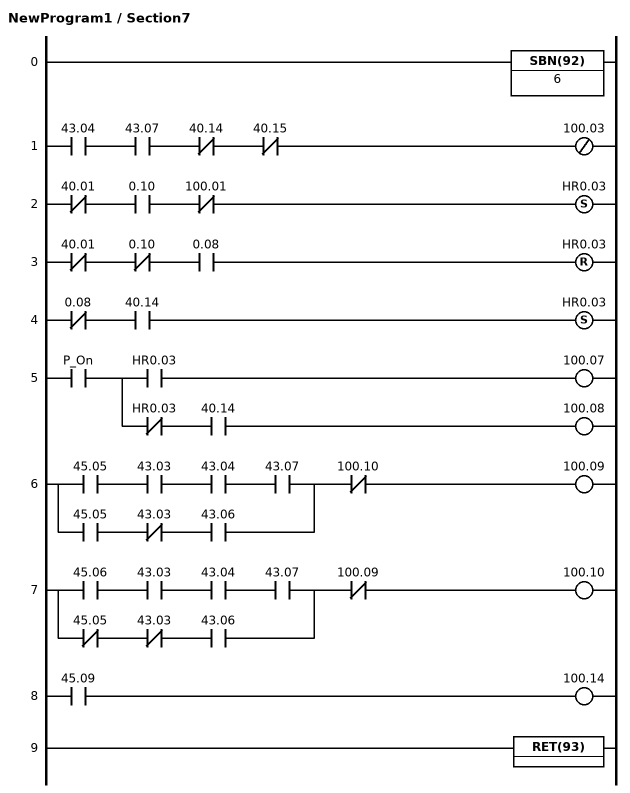
; [picture p24: NewProgram1 / Section7, rungs 0-9]
; rung 0
SBN(92) 6
; rung 1
LD 43.04
AND 43.07
ANDNOT 40.14
ANDNOT 40.15
OUTNOT 100.03
; rung 2
LDNOT 40.01
AND 0.10
ANDNOT 100.01
SET HR0.03
; rung 3
LDNOT 40.01
ANDNOT 0.10
AND 0.08
RSET HR0.03
; rung 4
LDNOT 0.08
AND 40.14
SET HR0.03
; rung 5
LD P_On
OUT TR0
AND HR0.03
OUT 100.07
LD TR0
ANDNOT HR0.03
AND 40.14
OUT 100.08
; rung 6
LD 45.05
AND 43.03
AND 43.04
AND 43.07
LD 45.05
ANDNOT 43.03
AND 43.06
ORLD
ANDNOT 100.10
OUT 100.09
; rung 7
LD 45.06
AND 43.03
AND 43.04
AND 43.07
LDNOT 45.05
ANDNOT 43.03
AND 43.06
ORLD
ANDNOT 100.09
OUT 100.10
; rung 8
LD 45.09
OUT 100.14
; rung 9
RET(93)

### Section Section8

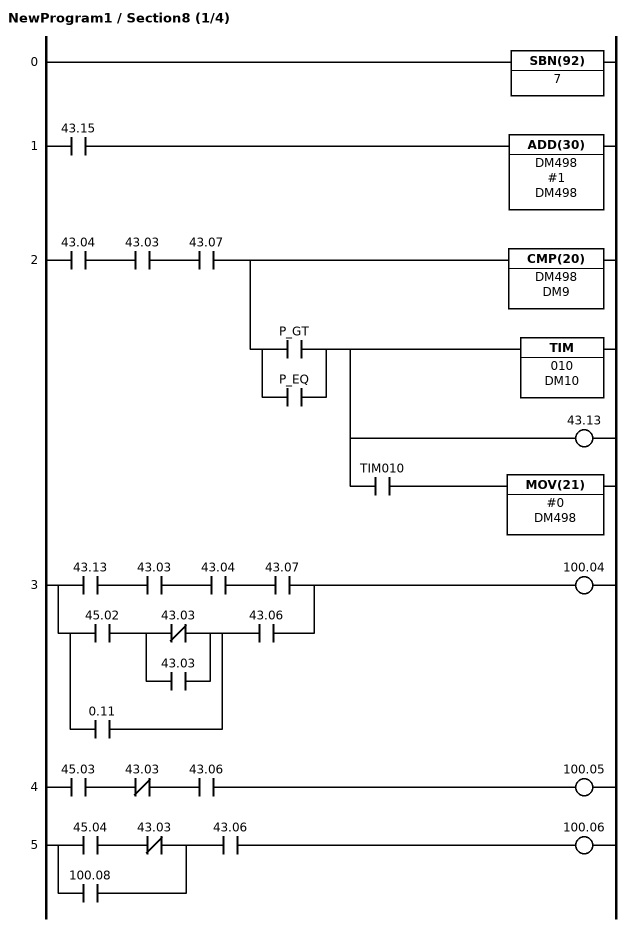
; rung 0
SBN(92) 7
; rung 1
LD 43.15
ADD(30) DM498 #1 DM498
; rung 2
LD 43.04
AND 43.03
AND 43.07
CMP(20) DM498 DM9
LD P_GT
OR P_EQ
ANDLD
TIM 010 DM10
OUT 43.13
AND TIM010
MOV(21) #0 DM498
; rung 3
LD 43.13
AND 43.03
AND 43.04
AND 43.07
LD 45.02
LDNOT 43.03
OR 43.03
ANDLD
OR 0.11
AND 43.06
ORLD
OUT 100.04
; rung 4
LD 45.03
ANDNOT 43.03
AND 43.06
OUT 100.05
; rung 5
LD 45.04
ANDNOT 43.03
OR 100.08
AND 43.06
OUT 100.06

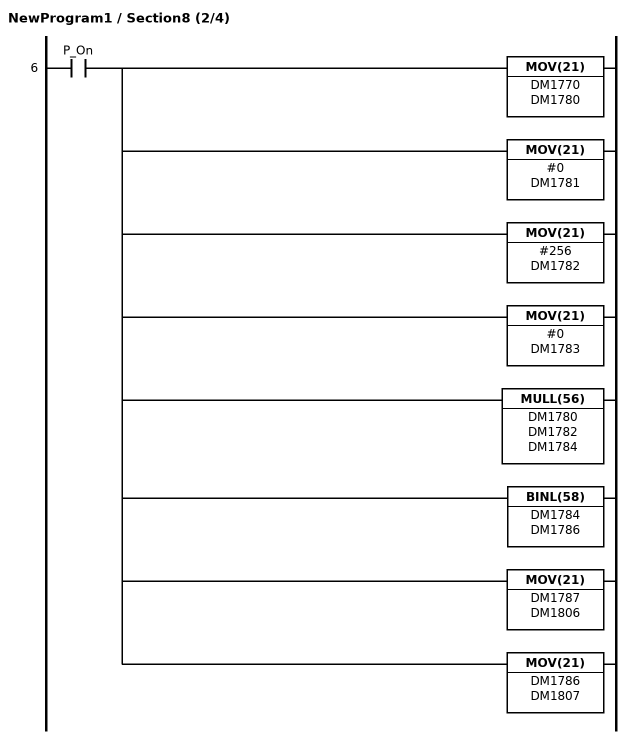
; rung 6
LD P_On
MOV(21) DM1770 DM1780
MOV(21) #0 DM1781
MOV(21) #256 DM1782
MOV(21) #0 DM1783
MULL(56) DM1780 DM1782 DM1784
BINL(58) DM1784 DM1786
MOV(21) DM1787 DM1806
MOV(21) DM1786 DM1807

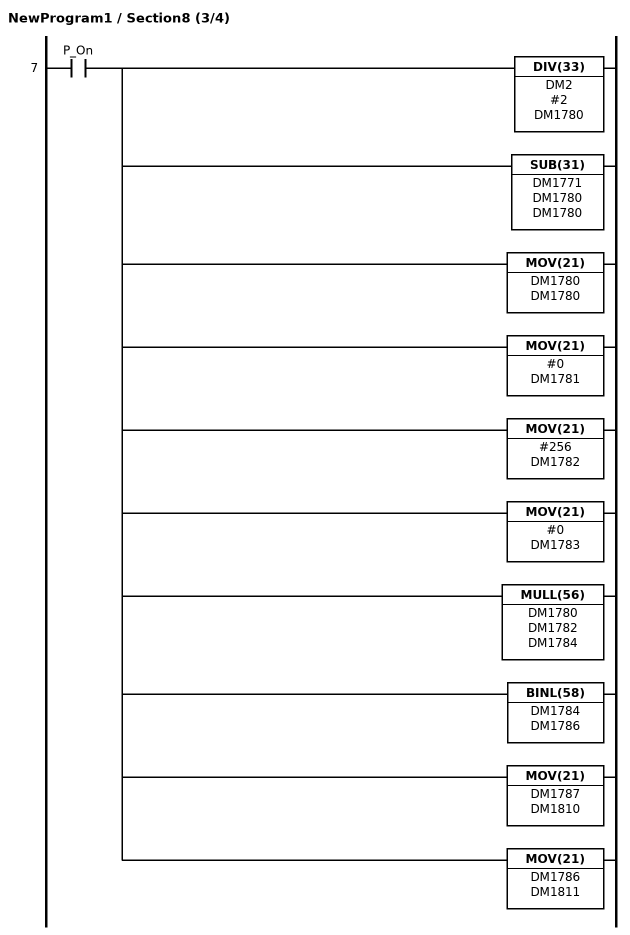
; rung 7
LD P_On
DIV(33) DM2 #2 DM1780
SUB(31) DM1771 DM1780 DM1780
MOV(21) DM1780 DM1780
MOV(21) #0 DM1781
MOV(21) #256 DM1782
MOV(21) #0 DM1783
MULL(56) DM1780 DM1782 DM1784
BINL(58) DM1784 DM1786
MOV(21) DM1787 DM1810
MOV(21) DM1786 DM1811

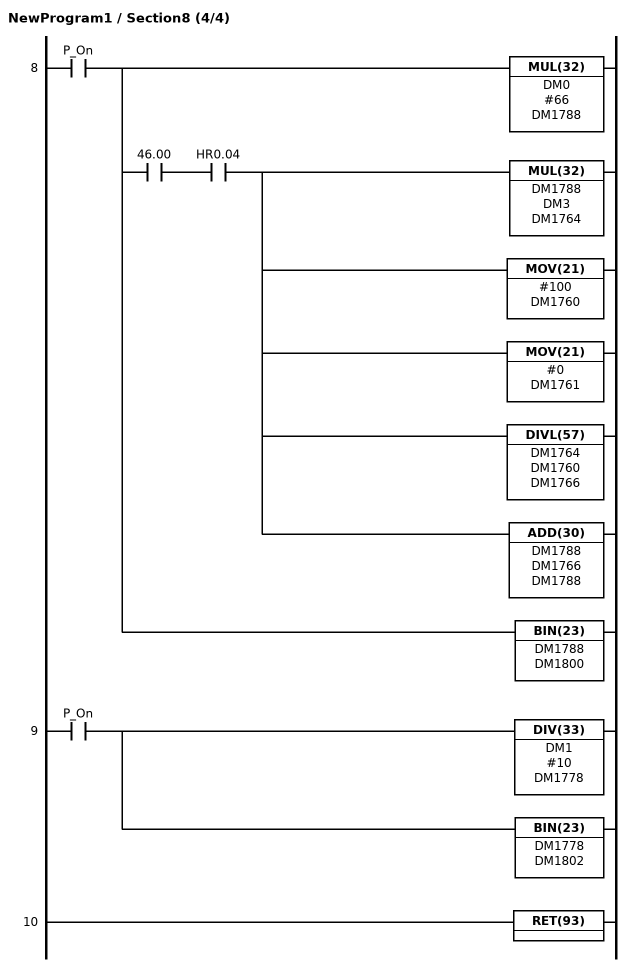
; rung 8
LD P_On
OUT TR0
MUL(32) DM0 #66 DM1788
AND 46.00
AND HR0.04
MUL(32) DM1788 DM3 DM1764
MOV(21) #100 DM1760
MOV(21) #0 DM1761
DIVL(57) DM1764 DM1760 DM1766
ADD(30) DM1788 DM1766 DM1788
LD TR0
BIN(23) DM1788 DM1800
; rung 9
LD P_On
DIV(33) DM1 #10 DM1778
BIN(23) DM1778 DM1802
; rung 10
RET(93)

### Section Section9

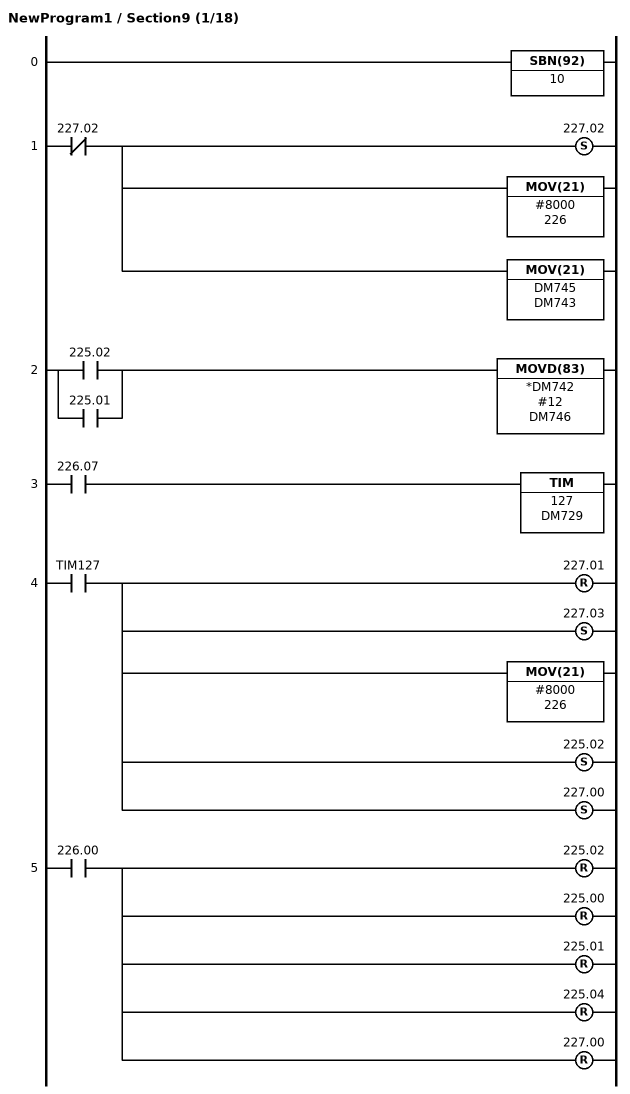
; rung 0
SBN(92) 10
; rung 1
LDNOT 227.02
SET 227.02
MOV(21) #8000 226
MOV(21) DM745 DM743
; rung 2
LD 225.02
OR 225.01
MOVD(83) *DM742 #12 DM746
; rung 3
LD 226.07
TIM 127 DM729
; rung 4
LD TIM127
RSET 227.01
SET 227.03
MOV(21) #8000 226
SET 225.02
SET 227.00
; rung 5
LD 226.00
RSET 225.02
RSET 225.00
RSET 225.01
RSET 225.04
RSET 227.00

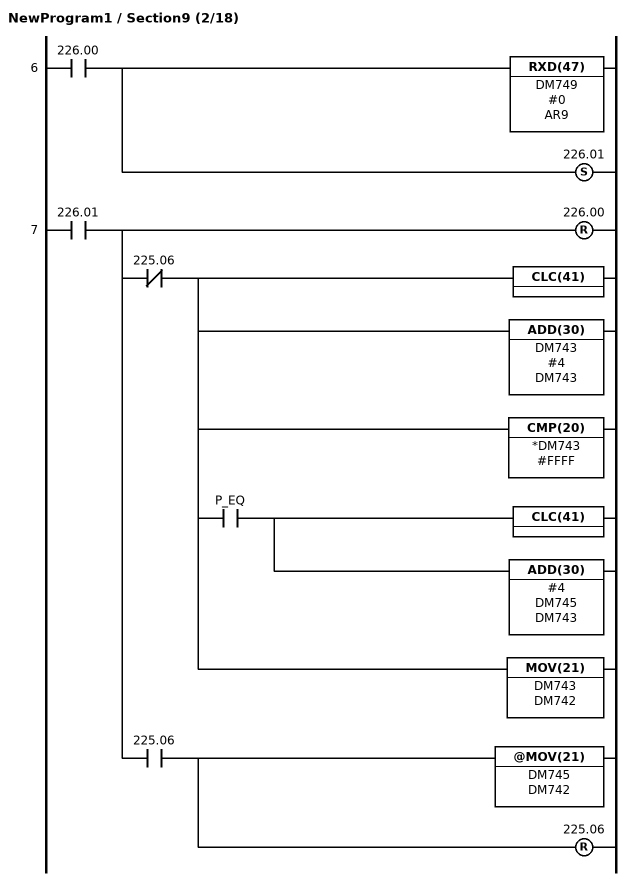
; rung 6
LD 226.00
RXD(47) DM749 #0 AR9
SET 226.01
; rung 7
LD 226.01
OUT TR0
RSET 226.00
ANDNOT 225.06
OUT TR1
CLC(41)
ADD(30) DM743 #4 DM743
CMP(20) *DM743 #FFFF
AND P_EQ
CLC(41)
ADD(30) #4 DM745 DM743
LD TR1
MOV(21) DM743 DM742
LD TR0
AND 225.06
@MOV(21) DM745 DM742
RSET 225.06

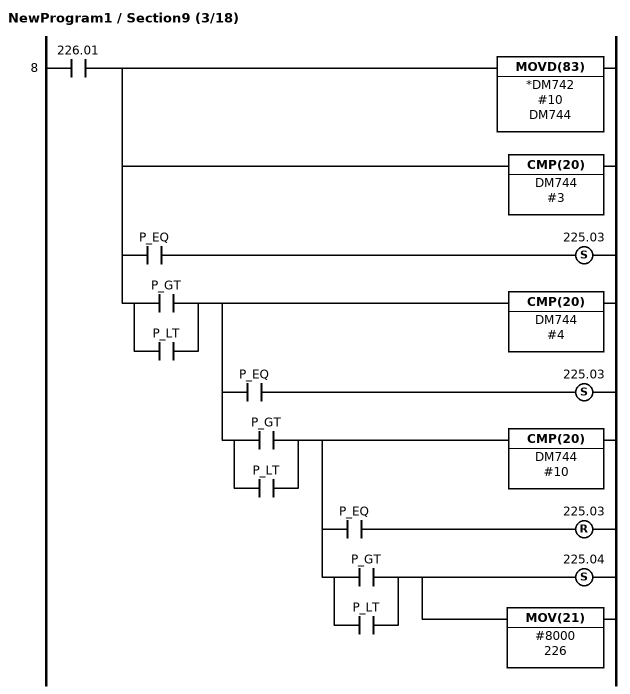
; rung 8
LD 226.01
OUT TR0
MOVD(83) *DM742 #10 DM744
CMP(20) DM744 #3
AND P_EQ
SET 225.03
LD TR0
LD P_GT
OR P_LT
ANDLD
OUT TR0
CMP(20) DM744 #4
AND P_EQ
SET 225.03
LD TR0
LD P_GT
OR P_LT
ANDLD
OUT TR0
CMP(20) DM744 #10
AND P_EQ
RSET 225.03
LD TR0
LD P_GT
OR P_LT
ANDLD
SET 225.04
MOV(21) #8000 226

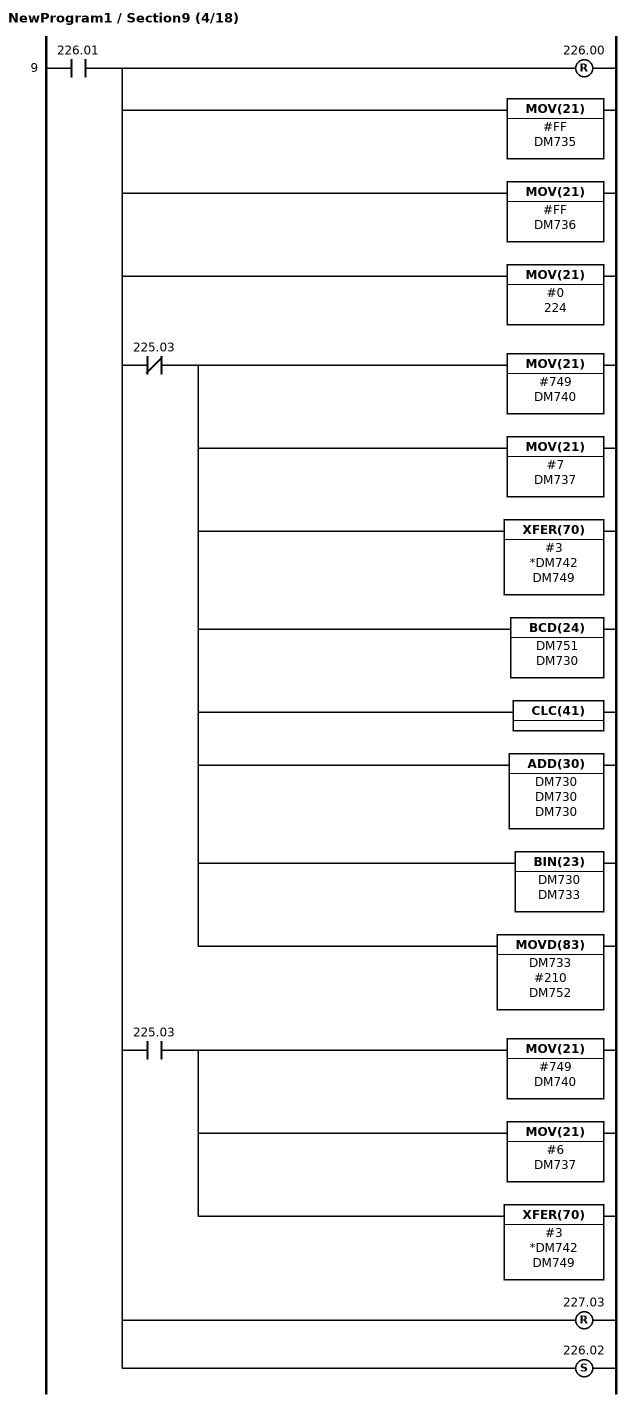
; rung 9
LD 226.01
OUT TR0
RSET 226.00
MOV(21) #FF DM735
MOV(21) #FF DM736
MOV(21) #0 224
ANDNOT 225.03
MOV(21) #749 DM740
MOV(21) #7 DM737
XFER(70) #3 *DM742 DM749
BCD(24) DM751 DM730
CLC(41)
ADD(30) DM730 DM730 DM730
BIN(23) DM730 DM733
MOVD(83) DM733 #210 DM752
LD TR0
AND 225.03
MOV(21) #749 DM740
MOV(21) #6 DM737
XFER(70) #3 *DM742 DM749
LD TR0
RSET 227.03
SET 226.02

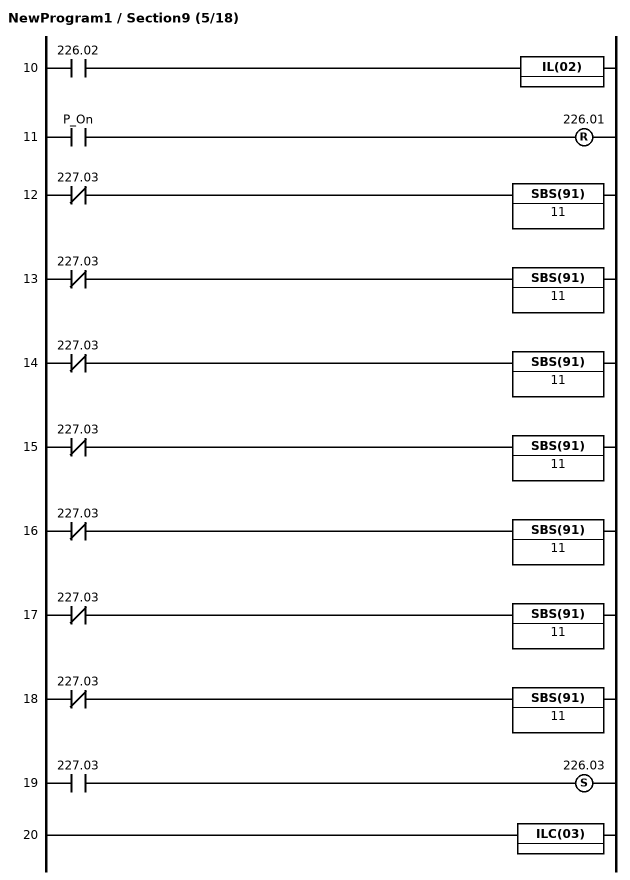
; rung 10
LD 226.02
IL(02)
; rung 11
LD P_On
RSET 226.01
; rung 12
LDNOT 227.03
SBS(91) 11
; rung 13
LDNOT 227.03
SBS(91) 11
; rung 14
LDNOT 227.03
SBS(91) 11
; rung 15
LDNOT 227.03
SBS(91) 11
; rung 16
LDNOT 227.03
SBS(91) 11
; rung 17
LDNOT 227.03
SBS(91) 11
; rung 18
LDNOT 227.03
SBS(91) 11
; rung 19
LD 227.03
SET 226.03
; rung 20
ILC(03)

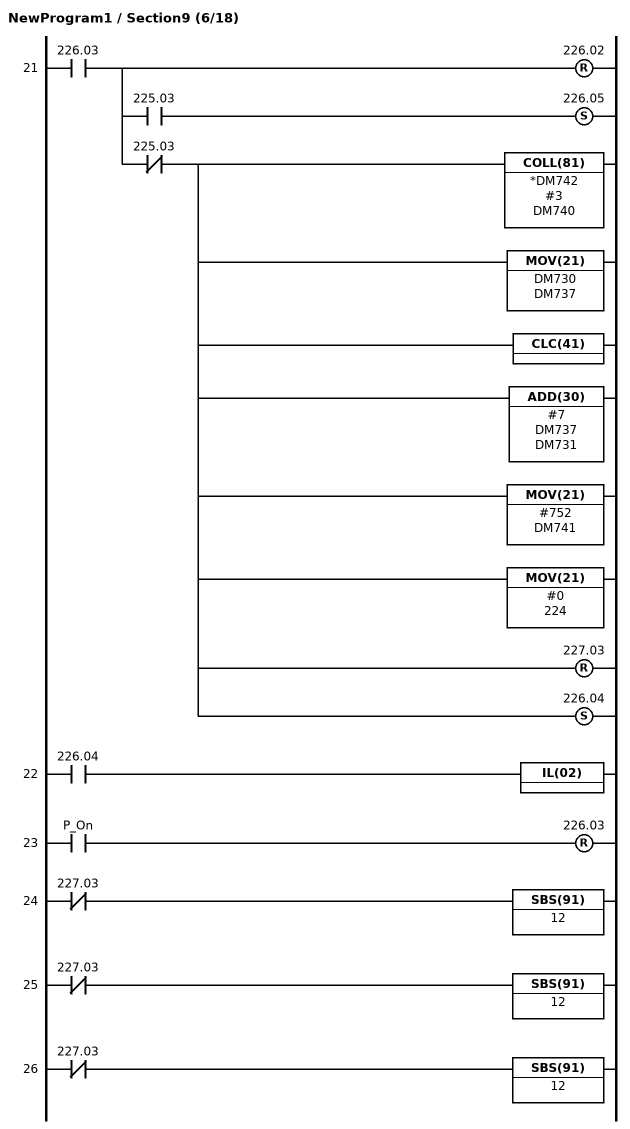
; rung 21
LD 226.03
OUT TR0
RSET 226.02
AND 225.03
SET 226.05
LD TR0
ANDNOT 225.03
COLL(81) *DM742 #3 DM740
MOV(21) DM730 DM737
CLC(41)
ADD(30) #7 DM737 DM731
MOV(21) #752 DM741
MOV(21) #0 224
RSET 227.03
SET 226.04
; rung 22
LD 226.04
IL(02)
; rung 23
LD P_On
RSET 226.03
; rung 24
LDNOT 227.03
SBS(91) 12
; rung 25
LDNOT 227.03
SBS(91) 12
; rung 26
LDNOT 227.03
SBS(91) 12

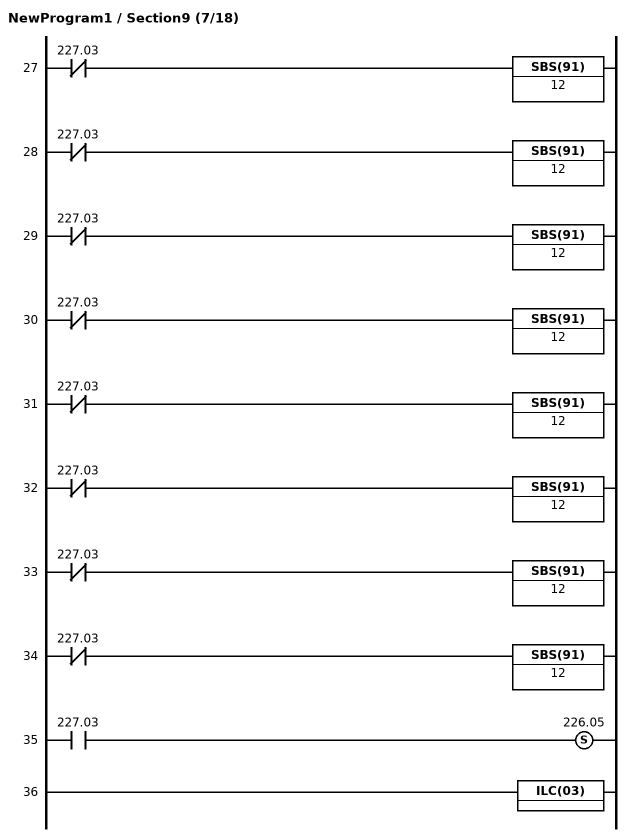
; rung 27
LDNOT 227.03
SBS(91) 12
; rung 28
LDNOT 227.03
SBS(91) 12
; rung 29
LDNOT 227.03
SBS(91) 12
; rung 30
LDNOT 227.03
SBS(91) 12
; rung 31
LDNOT 227.03
SBS(91) 12
; rung 32
LDNOT 227.03
SBS(91) 12
; rung 33
LDNOT 227.03
SBS(91) 12
; rung 34
LDNOT 227.03
SBS(91) 12
; rung 35
LD 227.03
SET 226.05
; rung 36
ILC(03)

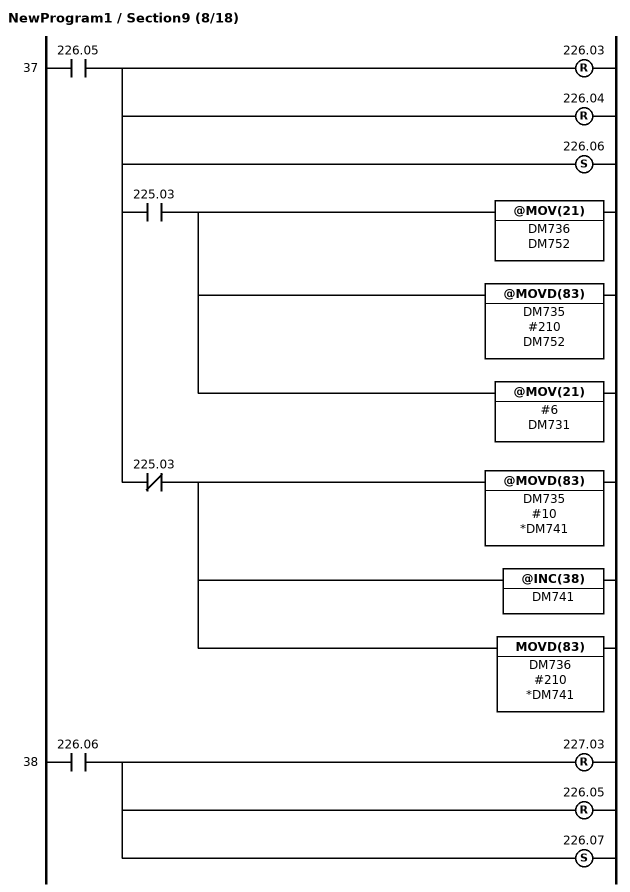
; rung 37
LD 226.05
OUT TR0
RSET 226.03
RSET 226.04
SET 226.06
AND 225.03
@MOV(21) DM736 DM752
@MOVD(83) DM735 #210 DM752
@MOV(21) #6 DM731
LD TR0
ANDNOT 225.03
@MOVD(83) DM735 #10 *DM741
@INC(38) DM741
MOVD(83) DM736 #210 *DM741
; rung 38
LD 226.06
RSET 227.03
RSET 226.05
SET 226.07

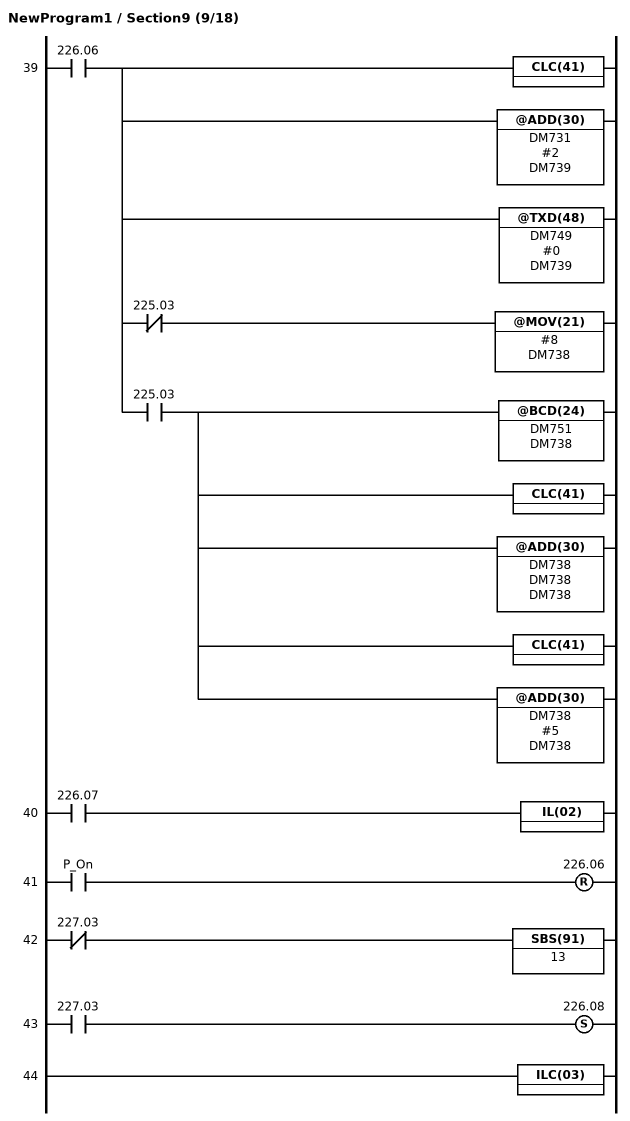
; rung 39
LD 226.06
OUT TR0
CLC(41)
@ADD(30) DM731 #2 DM739
@TXD(48) DM749 #0 DM739
ANDNOT 225.03
@MOV(21) #8 DM738
LD TR0
AND 225.03
@BCD(24) DM751 DM738
CLC(41)
@ADD(30) DM738 DM738 DM738
CLC(41)
@ADD(30) DM738 #5 DM738
; rung 40
LD 226.07
IL(02)
; rung 41
LD P_On
RSET 226.06
; rung 42
LDNOT 227.03
SBS(91) 13
; rung 43
LD 227.03
SET 226.08
; rung 44
ILC(03)

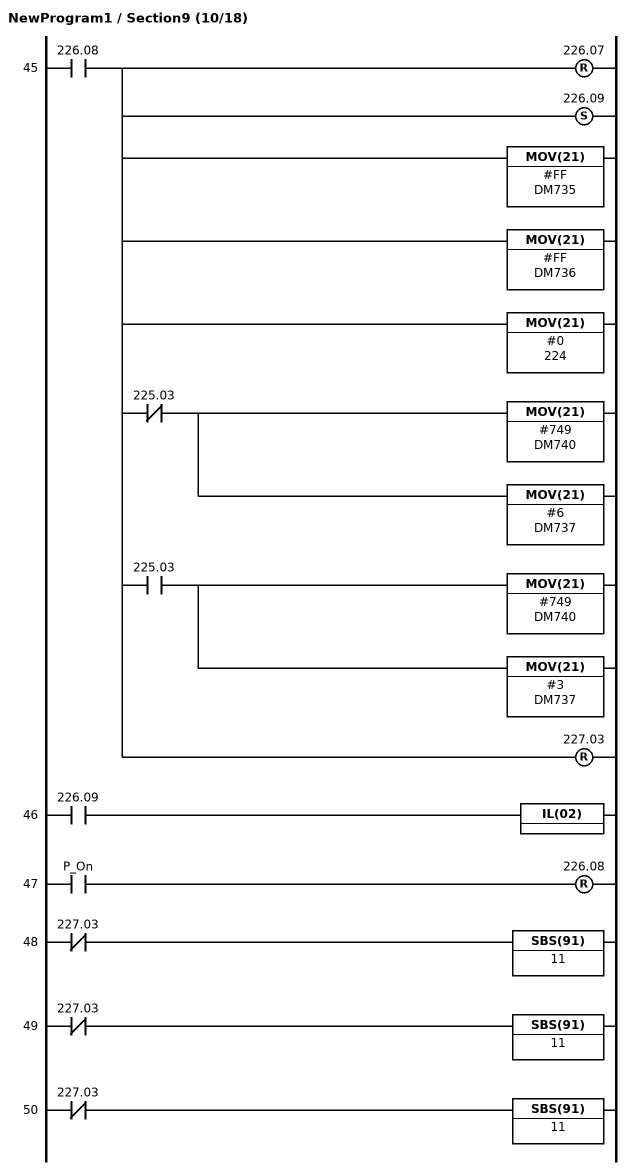
; rung 45
LD 226.08
OUT TR0
RSET 226.07
SET 226.09
MOV(21) #FF DM735
MOV(21) #FF DM736
MOV(21) #0 224
ANDNOT 225.03
MOV(21) #749 DM740
MOV(21) #6 DM737
LD TR0
AND 225.03
MOV(21) #749 DM740
MOV(21) #3 DM737
LD TR0
RSET 227.03
; rung 46
LD 226.09
IL(02)
; rung 47
LD P_On
RSET 226.08
; rung 48
LDNOT 227.03
SBS(91) 11
; rung 49
LDNOT 227.03
SBS(91) 11
; rung 50
LDNOT 227.03
SBS(91) 11

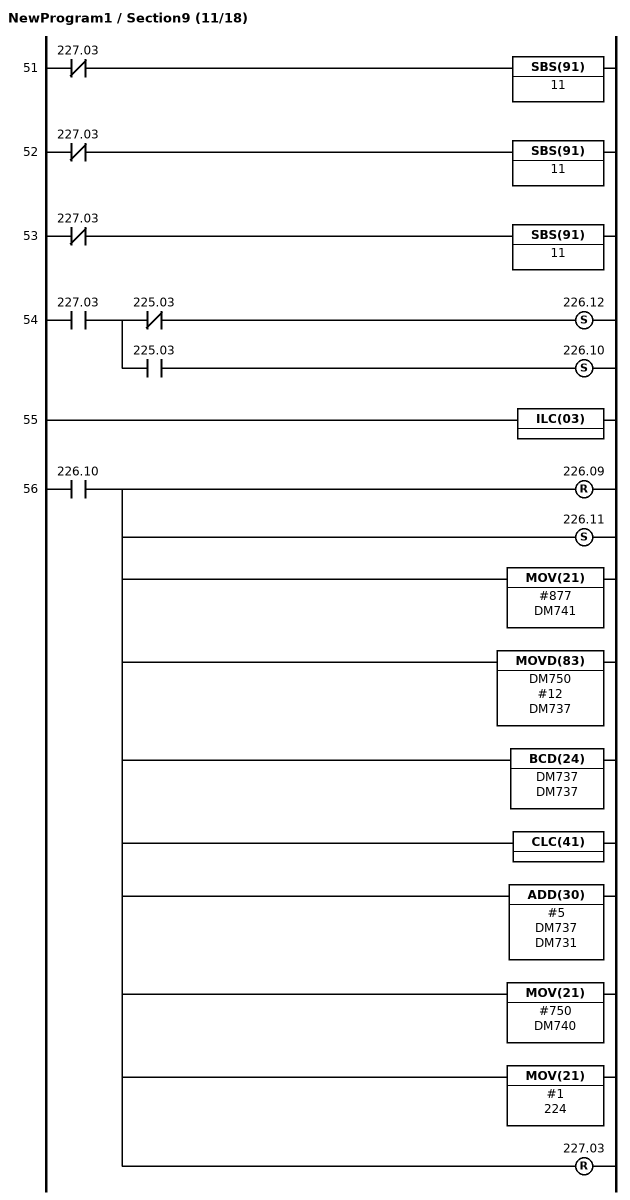
; rung 51
LDNOT 227.03
SBS(91) 11
; rung 52
LDNOT 227.03
SBS(91) 11
; rung 53
LDNOT 227.03
SBS(91) 11
; rung 54
LD 227.03
OUT TR0
ANDNOT 225.03
SET 226.12
LD TR0
AND 225.03
SET 226.10
; rung 55
ILC(03)
; rung 56
LD 226.10
RSET 226.09
SET 226.11
MOV(21) #877 DM741
MOVD(83) DM750 #12 DM737
BCD(24) DM737 DM737
CLC(41)
ADD(30) #5 DM737 DM731
MOV(21) #750 DM740
MOV(21) #1 224
RSET 227.03

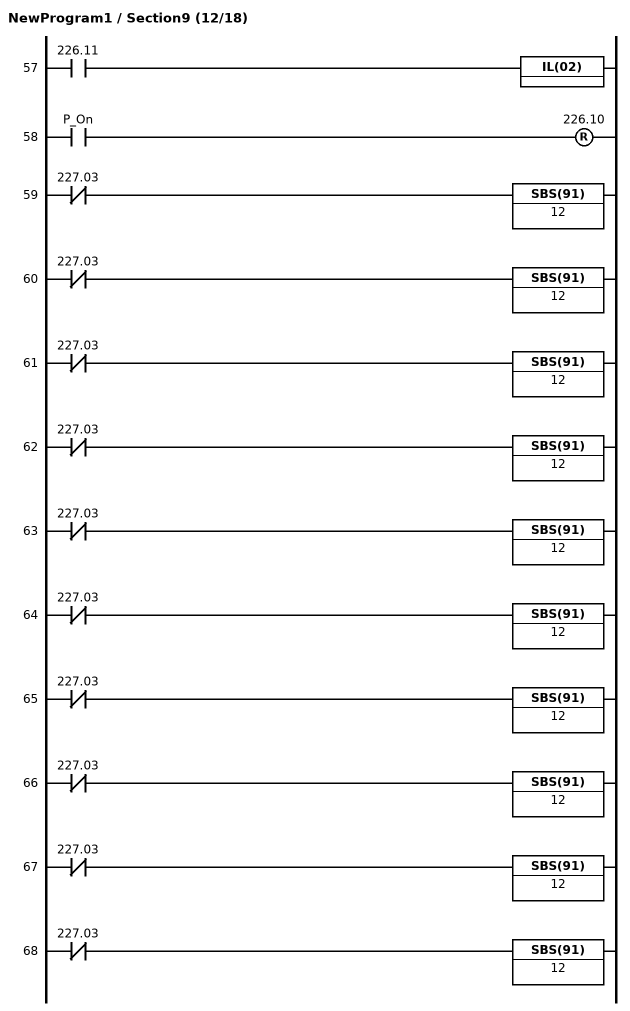
; rung 57
LD 226.11
IL(02)
; rung 58
LD P_On
RSET 226.10
; rung 59
LDNOT 227.03
SBS(91) 12
; rung 60
LDNOT 227.03
SBS(91) 12
; rung 61
LDNOT 227.03
SBS(91) 12
; rung 62
LDNOT 227.03
SBS(91) 12
; rung 63
LDNOT 227.03
SBS(91) 12
; rung 64
LDNOT 227.03
SBS(91) 12
; rung 65
LDNOT 227.03
SBS(91) 12
; rung 66
LDNOT 227.03
SBS(91) 12
; rung 67
LDNOT 227.03
SBS(91) 12
; rung 68
LDNOT 227.03
SBS(91) 12

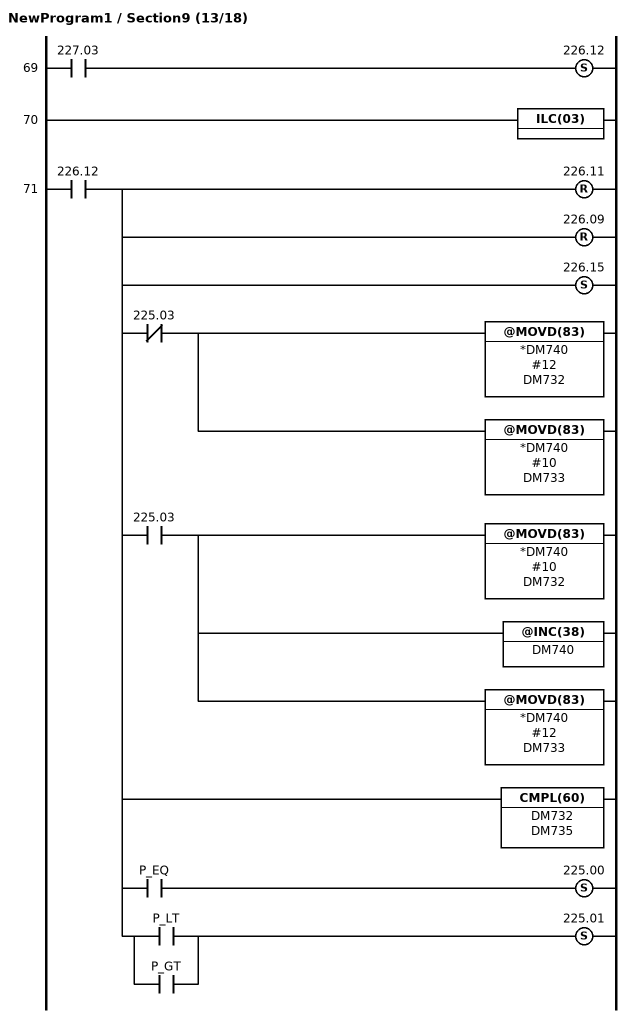
; rung 69
LD 227.03
SET 226.12
; rung 70
ILC(03)
; rung 71
LD 226.12
OUT TR0
RSET 226.11
RSET 226.09
SET 226.15
ANDNOT 225.03
@MOVD(83) *DM740 #12 DM732
@MOVD(83) *DM740 #10 DM733
LD TR0
AND 225.03
@MOVD(83) *DM740 #10 DM732
@INC(38) DM740
@MOVD(83) *DM740 #12 DM733
LD TR0
CMPL(60) DM732 DM735
AND P_EQ
SET 225.00
LD TR0
LD P_LT
OR P_GT
ANDLD
SET 225.01

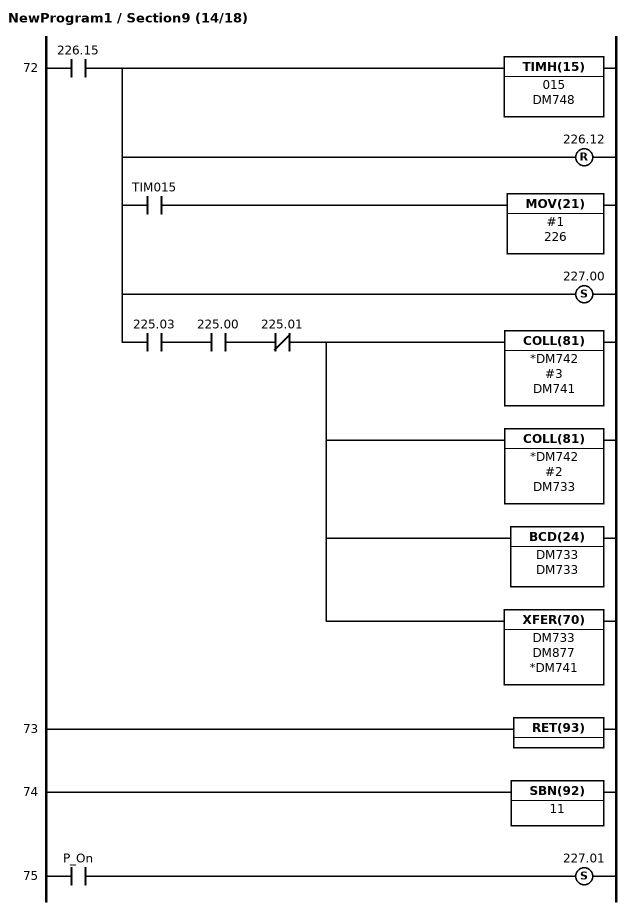
; rung 72
LD 226.15
OUT TR0
TIMH(15) 015 DM748
RSET 226.12
AND TIM015
MOV(21) #1 226
LD TR0
SET 227.00
AND 225.03
AND 225.00
ANDNOT 225.01
COLL(81) *DM742 #3 DM741
COLL(81) *DM742 #2 DM733
BCD(24) DM733 DM733
XFER(70) DM733 DM877 *DM741
; rung 73
RET(93)
; rung 74
SBN(92) 11
; rung 75
LD P_On
SET 227.01

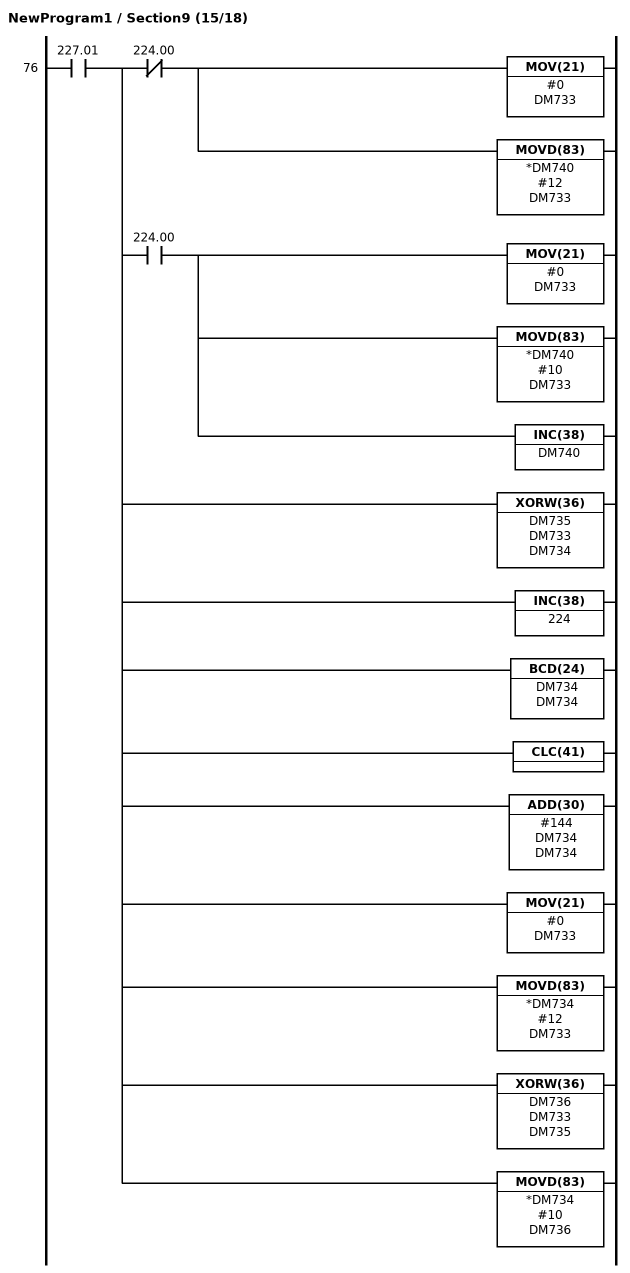
; rung 76
LD 227.01
OUT TR0
ANDNOT 224.00
MOV(21) #0 DM733
MOVD(83) *DM740 #12 DM733
LD TR0
AND 224.00
MOV(21) #0 DM733
MOVD(83) *DM740 #10 DM733
INC(38) DM740
LD TR0
XORW(36) DM735 DM733 DM734
INC(38) 224
BCD(24) DM734 DM734
CLC(41)
ADD(30) #144 DM734 DM734
MOV(21) #0 DM733
MOVD(83) *DM734 #12 DM733
XORW(36) DM736 DM733 DM735
MOVD(83) *DM734 #10 DM736

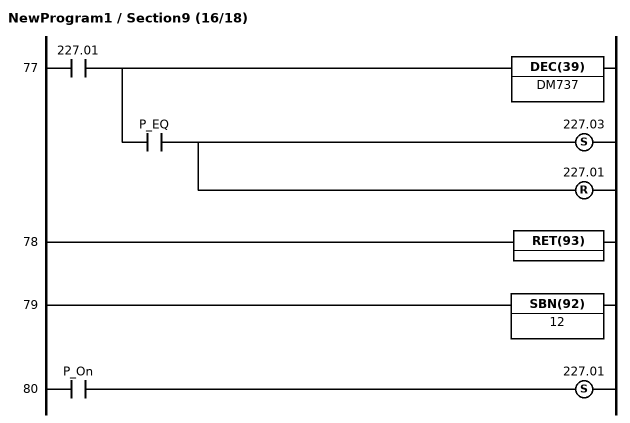
; rung 77
LD 227.01
DEC(39) DM737
AND P_EQ
SET 227.03
RSET 227.01
; rung 78
RET(93)
; rung 79
SBN(92) 12
; rung 80
LD P_On
SET 227.01

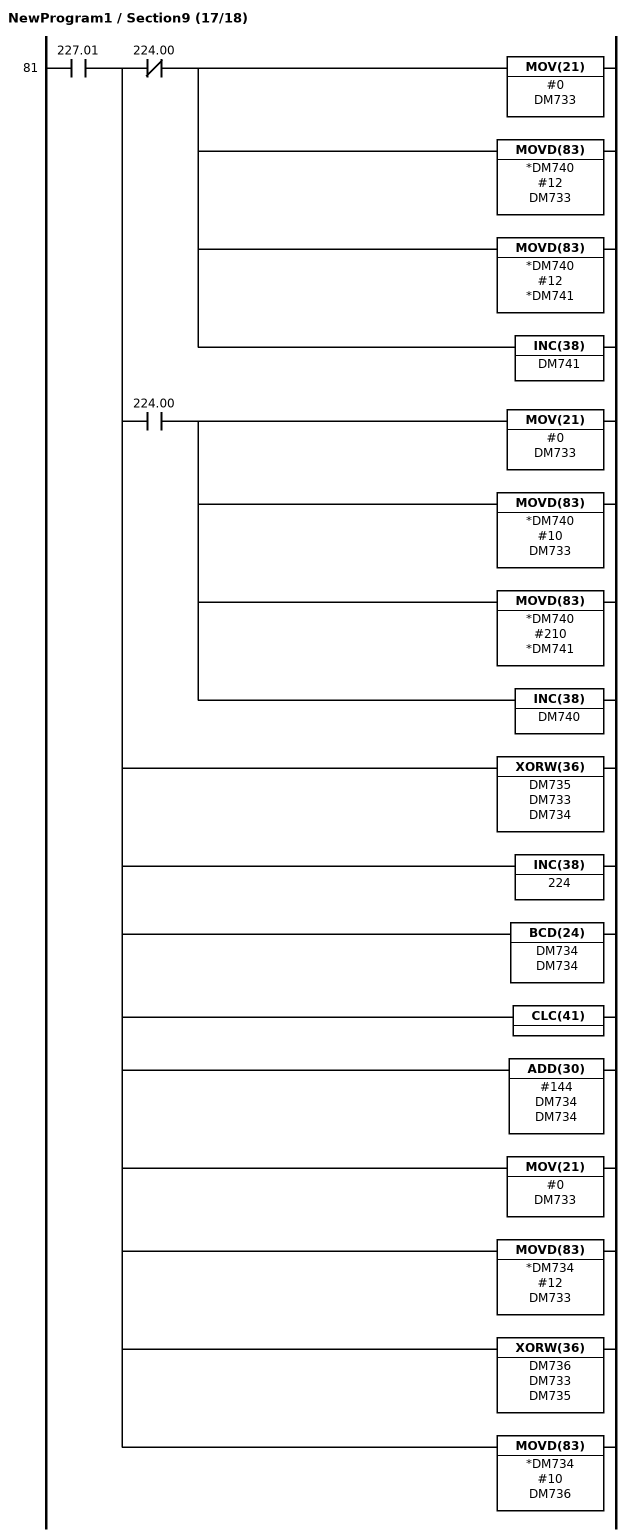
; rung 81
LD 227.01
OUT TR0
ANDNOT 224.00
MOV(21) #0 DM733
MOVD(83) *DM740 #12 DM733
MOVD(83) *DM740 #12 *DM741
INC(38) DM741
LD TR0
AND 224.00
MOV(21) #0 DM733
MOVD(83) *DM740 #10 DM733
MOVD(83) *DM740 #210 *DM741
INC(38) DM740
LD TR0
XORW(36) DM735 DM733 DM734
INC(38) 224
BCD(24) DM734 DM734
CLC(41)
ADD(30) #144 DM734 DM734
MOV(21) #0 DM733
MOVD(83) *DM734 #12 DM733
XORW(36) DM736 DM733 DM735
MOVD(83) *DM734 #10 DM736

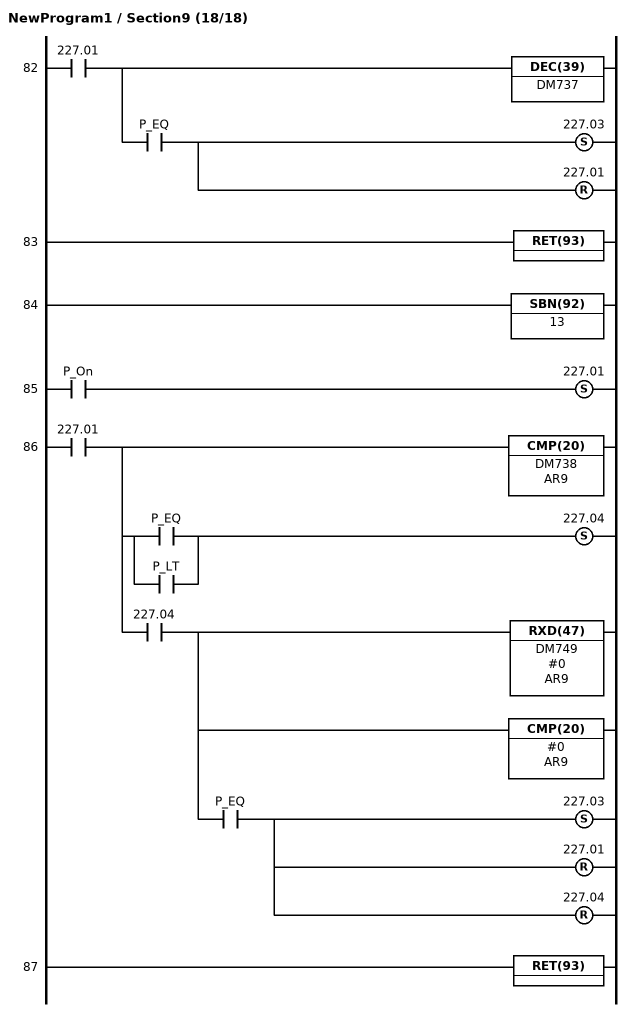
; rung 82
LD 227.01
DEC(39) DM737
AND P_EQ
SET 227.03
RSET 227.01
; rung 83
RET(93)
; rung 84
SBN(92) 13
; rung 85
LD P_On
SET 227.01
; rung 86
LD 227.01
OUT TR0
CMP(20) DM738 AR9
LD P_EQ
OR P_LT
ANDLD
SET 227.04
LD TR0
AND 227.04
RXD(47) DM749 #0 AR9
CMP(20) #0 AR9
AND P_EQ
SET 227.03
RSET 227.01
RSET 227.04
; rung 87
RET(93)

### Section Section10
; rung 0
END(01)